PROGRAM MobjectCollectionsExample
VAR
END_VAR

END_PROGRAM

(* stored: Version 1.1.0.1, ProductVersion 3.1.4024.13
   POU MobjectCollectionsExample: Id {44aca389-efe5-0491-162d-4e37ca5d5fd8}, SpecialFunc None *)
